{attribute 'reflection'} 
FUNCTION_BLOCK FB_DigitalOutput IMPLEMENTS I_DigitalChannel
VAR_INPUT
END_VAR
VAR_OUTPUT
END_VAR
VAR
	sIdentifier:				STRING(25);		// Equipment ID
	Channel			AT%Q*: BOOL;	// Link to output
END_VAR

// https://github.com/PeterZerlauth/Tc3_Component

PROPERTY PUBLIC P_ID : STRING(25)
GET
P_ID:= sIdentifier;
END_GET
END_PROPERTY

PROPERTY P_State : EPlcMappingStatus
GET
P_State:= F_GetMappingStatus(adr(Channel), sizeof(BOOL));
END_GET
END_PROPERTY

PROPERTY PUBLIC P_Value : bool
GET
P_Value:= Channel;
END_GET
SET // PUBLIC
Channel:= P_Value;
END_SET
END_PROPERTY

END_FUNCTION_BLOCK

(* stored: Version 1.1.0.1
   POU FB_DigitalOutput: Id {9c6c856c-bfc6-09b8-0205-5829241d18e2}, SpecialFunc None
   Property P_ID: Id {f50a731d-33e5-019b-0fc3-26d5f1374f48}
   Get Get: Id {cfa231bf-ff32-0ded-1b81-f9ced6eebfc5}
   Property P_State: Id {828aeade-e2eb-0b55-3817-3951b800d035}
   Get Get: Id {3e020151-e801-097e-31b7-4a7cc9867898}
   Property P_Value: Id {696506a3-db60-0746-2f1d-1c14b42d34db}
   Get Get: Id {fde9f4b6-16df-028f-2ce8-9cfbd063a439}
   Set Set: Id {69af308d-96e0-0ca6-0d1c-c75ab3a009fc} *)
